FUNCTION Keyence_LRTB2000C : REAL
VAR_INPUT
	Byte0 : BYTE;
	Byte1 : BYTE;
END_VAR

VAR
END_VAR


Keyence_LRTB2000C := Byte0*256 + Byte1;

END_FUNCTION

(* stored: Version 1.1.0.1, ProductVersion 3.1.4024.11
   POU Keyence_LRTB2000C: Id {dc2950e0-5829-4e9f-9b8f-f4628010470a}, SpecialFunc None *)
